{attribute 'qualified_only' := ''}
{attribute 'strict' := ''}
TYPE MC_BUFFER_MODE :
(
	mcAborting := 0,
	mcBuffered := 1,
	mcBlendingLow := 2,
	mcBlendingPrevious := 3,
	mcBlendingNext := 4,
	mcBlendingHigh := 5
);
END_TYPE

(* stored: Version 1.1.0.1, ProductVersion 3.1.4024.12
   DUT MC_BUFFER_MODE: Id {3ed947d8-b908-4b41-a79d-f94b16833959} *)
